{attribute 'pack_mode' := '1'}
    {attribute 'OPC.UA.DA' := '1'}
    {attribute 'OPC.UA.DA.StructuredType' := '1'}
    (*
    ST_RWInterlock_HMI_IgnitionExp
    ==================================================
    Generated from Ignition UDT: RW_Interlock_V2
    Total tags: 12
    Generated on: 2025-09-15 12:56:43
    *)
    TYPE ST_RWInterlock_HMI_IgnitionExp :
    STRUCT
        {attribute 'OPC.UA.DA' := '1'}
        {attribute 'OPC.UA.DA.Description' := 'Time delay before interlock trip is active'}
        // Time delay before interlock trip is active
        HMI_Cfg_IntlkOnDly : REAL := 0.0;
        {attribute 'OPC.UA.DA' := '1'}
        {attribute 'OPC.UA.DA.Access' := '1'}
        {attribute 'OPC.UA.DA.Description' := 'Packed bits to HMI'}
        // Packed bits to HMI
        S_HMIBits : DINT := 0;		// Read-only tag
        {attribute 'OPC.UA.DA' := '1'}
        {attribute 'OPC.UA.DA.Description' := '1=Only Maint can reset this Interlock'}
        // 1=Only Maint can reset this Interlock
        UDT_mem_MaintOnlyReset : BOOL := FALSE;
        {attribute 'OPC.UA.DA' := '1'}
        {attribute 'OPC.UA.DA.Access' := '1'}
        {attribute 'OPC.UA.DA.Description' := 'NonBypassable Interlock Status (1=Tripped, 0=OK to run)'}
        // NonBypassable Interlock Status (1=Tripped, 0=OK to run)
        S_NBIntlkTripped : BOOL := FALSE;		// Read-only tag
        {attribute 'OPC.UA.DA' := '1'}
        {attribute 'OPC.UA.DA.Access' := '1'}
        {attribute 'OPC.UA.DA.Description' := 'Interlock Status (1=Tripped, 0=OK to run)'}
        // Interlock Status (1=Tripped, 0=OK to run)
        S_Tripped : BOOL := FALSE;		// Read-only tag

        {attribute 'OPC.UA.DA' := '1'}
        {attribute 'OPC.UA.DA.Description' := 'Minimum time for the output to be held true to verify HMI receives status'}
        // Minimum time for the output to be held true to verify HMI receives ...
        HMI_Cfg_IntlkOffDly : REAL := 0.0;
        {attribute 'OPC.UA.DA' := '1'}
        {attribute 'OPC.UA.DA.Description' := '1= Bypass Interlocked Tripped condition, Enabled'}
        // 1= Bypass Interlocked Tripped condition, Enabled
        HMI_C_Bypass : BOOL := FALSE;
        {attribute 'OPC.UA.DA' := '1'}
        {attribute 'OPC.UA.DA.Description' := 'Reset Command'}
        // Reset Command
        HMI_C_Reset : BOOL := FALSE;
        {attribute 'OPC.UA.DA' := '1'}
        {attribute 'OPC.UA.DA.Access' := '1'}
        {attribute 'OPC.UA.DA.Description' := '1=Interlock condition can be bypassed'}
        // 1=Interlock condition can be bypassed
        Cfg_Bypassable : BOOL := FALSE;		// Read-only tag
        {attribute 'OPC.UA.DA' := '1'}
        {attribute 'OPC.UA.DA.Access' := '1'}
        {attribute 'OPC.UA.DA.Description' := 'Bypass function is enabled by Maint/Eng'}
        // Bypass function is enabled by Maint/Eng
        S_BypEnabled : BOOL := FALSE;		// Read-only tag

        {attribute 'OPC.UA.DA' := '1'}
        {attribute 'OPC.UA.DA.Access' := '1'}
        {attribute 'OPC.UA.DA.Description' := '1= Interlock is latched (sealed in) and requires reset'}
        // 1= Interlock is latched (sealed in) and requires reset
        Cfg_Latched : BOOL := FALSE;		// Read-only tag
        {attribute 'OPC.UA.DA' := '1'}
        {attribute 'OPC.UA.DA.Access' := '1'}
        {attribute 'OPC.UA.DA.Description' := '1=Tripped or Interlock Condition, 0=OK to run'}
        // 1=Tripped or Interlock Condition, 0=OK to run
        C_Trip_Condition : BOOL := FALSE;		// Read-only tag
    END_STRUCT
    END_TYPE

(* stored: Version 1.1.0.1
   DUT ST_RWInterlock_HMI_IgnitionExp: Id {e0d82633-89d2-43a9-93d0-17ec2e42ab6f} *)
